Universal Robots PolyScope program: 2.10.2024.urp

Program 2.10.2024 (installation=default directory=/programs createdIn=3.15.8.106339 lastSavedIn=3.15.8.106339 robotSerialNumber=2023330214)
Calibrated DH parameters: a=[-0.000161, -0.243516, -0.175941, 0.000055, -0.000127, 0]; d=[0.151869, -0.926342, 57.568096, -56.529557, 0.085345, 0.082309]; alpha=[1.571543, -0.007517, 0.002128, 1.570286, -1.573097, 0]; deltaTheta=[0.000048, 0.028487, 0.571925, -0.600676, 0.000055, 0.000013]
BeforeStart
  p_12 := True
  Timer (action=Start) variable(name=timer_1)
  MoveJ speed 60 deg/s, acceleration 80 deg/s^2 (useActiveTCP=true)
    Waypoint Start: TCP in base x=-380.658 y=-285.177 z=13.926 mm, rx=-0.8605 ry=2.9837 rz=0.005 rad; joints [-128.616, -137.162, -81.807, -52.682, 90.828, -2230.513] deg; flange x=-351.756 y=-266.308 z=98.21 mm, rx=-0.8605 ry=2.9837 rz=0.005 rad
  p := Start
Robot Program (runOnlyOnce=false)
  Loop While (checkContinuously=true) expression=p_12
    Script: p[0]=p[0]+0.065
    MoveL speed 250 mm/s, acceleration 1200 mm/s^2 (useActiveTCP=true) feature=Base
      MoveDirectionNode (selectedDirection=ZMinus)
        Until DISTANCE (allowActions=false deceleration=3 distanceNodeType=STOP) Distance=0.022; motionParameters(blendRadius=0)
      MoveDirectionNode (selectedDirection=ZPlus)
        Until DISTANCE (allowActions=false deceleration=3 distanceNodeType=STOP) Distance=0.022; motionParameters(blendRadius=0)
      Waypoint Waypoint (Variable): variable=p
    Wait Sleep waitTime=1
    MoveL speed 250 mm/s, acceleration 1200 mm/s^2 (useActiveTCP=true) feature=Base
      Waypoint Waypoint (Variable): variable=p
Thread Thread_1 (runOnlyOnce=false)
  If timer_1>4
    Timer (action=Stop) variable=timer_1
    p_12 := False
    Popup Message (haltProgram=false message=premi per riavviare il robot inputType=Text)
    p_12 := True
    Timer (action=Start) variable=timer_1
    Timer (action=Reset) variable=timer_1
